
// ===== library: MasterCopy "Scale_current_output" =====

FUNCTION "Scale_current_output" : Void   // FC2, LAD
TITLE = Scale current output from 4-20 mA to 0-20 mA
{ S7_Optimized_Access := 'FALSE' }
VERSION : 0.1
// (27648-5530) 
// f(x) =  ------------------------- * x +5530 
//                 27648
   VAR_INPUT
      "r_output_4-20mA" : Real;
   END_VAR
   VAR_OUTPUT
      "w_output_0-20mA" : Word;
   END_VAR
   VAR_TEMP
      r_analog_ouput_temp : Real;
      r_factor : Real;
   END_VAR
BEGIN

REGION Network 1
   // multiply  by range  4-20mA ( 27648-5529,6=22118,4)
   // f(x1) = x * 22118
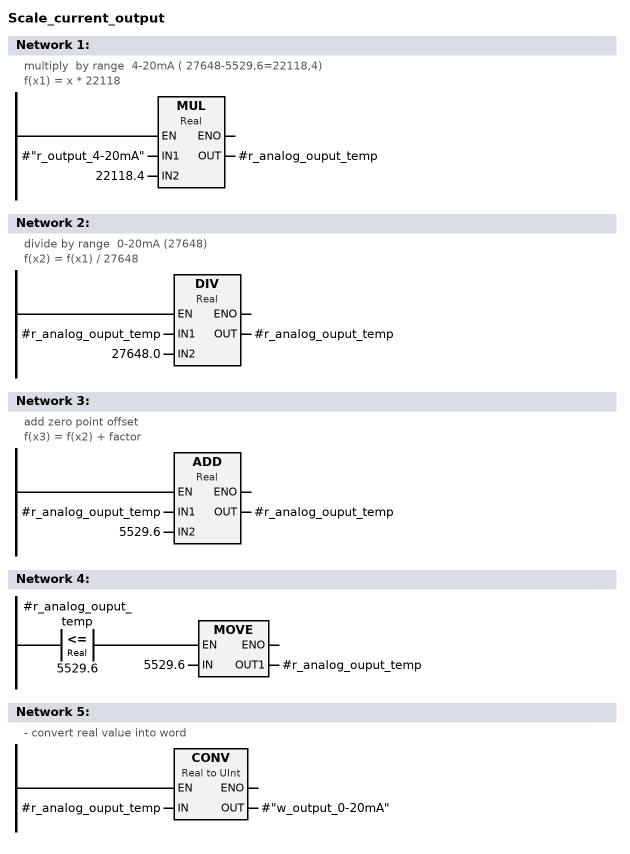
   RUNG wire#powerrail
      { S7_Templates := "SrcType := Real"; S7_GenerateENO := "TRUE" } Mul(in1 := #"r_output_4-20mA", in2 := 22118.4, out => #r_analog_ouput_temp)
   END_RUNG
   // the same network as SCL:
   #r_analog_ouput_temp := #"r_output_4-20mA" * 22118.4;
END_REGION

REGION Network 2
   // divide by range  0-20mA (27648)
   // f(x2) = f(x1) / 27648
   RUNG wire#powerrail
      { S7_Templates := "SrcType := Real"; S7_GenerateENO := "TRUE" } Div(in1 := #r_analog_ouput_temp, in2 := 27648.0, out => #r_analog_ouput_temp)
   END_RUNG
   // the same network as SCL:
   #r_analog_ouput_temp := #r_analog_ouput_temp / 27648.0;
END_REGION

REGION Network 3
   // add zero point offset
   // f(x3) = f(x2) + factor
   RUNG wire#powerrail
      { S7_Templates := "SrcType := Real"; S7_GenerateENO := "TRUE" } Add(in1 := #r_analog_ouput_temp, in2 := 5529.6, out => #r_analog_ouput_temp)
   END_RUNG
   // the same network as SCL:
   #r_analog_ouput_temp := #r_analog_ouput_temp + 5529.6;
END_REGION

REGION Network 4
   RUNG wire#powerrail
      { S7_Templates := "SrcType := Real" } LE_Contact(in1 := #r_analog_ouput_temp, in2 := 5529.6)
      { S7_GenerateENO := "TRUE" } Move(in := 5529.6, out1 => #r_analog_ouput_temp)
   END_RUNG
   // the same network as SCL:
   IF #r_analog_ouput_temp <= 5529.6 THEN #r_analog_ouput_temp := 5529.6; END_IF;
END_REGION

REGION Network 5
   // - convert real value into word
   RUNG wire#powerrail
      { S7_Templates := "[SrcType := Real, DestType := UInt]"; S7_GenerateENO := "TRUE" } Convert(in := #r_analog_ouput_temp, out => #"w_output_0-20mA")
   END_RUNG
   // the same network as SCL:
   #"w_output_0-20mA" := REAL_TO_UINT(#r_analog_ouput_temp);
END_REGION
END_FUNCTION

// ===== library: MasterCopy "Scale_current_input" =====

FUNCTION "Scale_current_input" : Void   // FC1, LAD
TITLE = Scale current input from 0-20 mA to 4-20 mA
{ S7_Optimized_Access := 'FALSE' }
VERSION : 0.1
// 27648
// f(x) =  ------------------------------- * x - 6912
//            (27648 - 5529,6)
   VAR_INPUT
      r_wire_break_limit : Real;
      "w_input_0-20mA" : Word;
   END_VAR
   VAR_OUTPUT
      b_wire_break : Bool;
      "r_input_4-20mA" : Real;
   END_VAR
   VAR_TEMP
      r_analog_input_temp : Real;
      r_factor : Real;
   END_VAR
   VAR_TEMP   // added for the SCL form of the ladder/FBD networks
      _w1 : Bool;
   END_VAR
BEGIN

REGION Network 1
   // - Convert analog  value to real
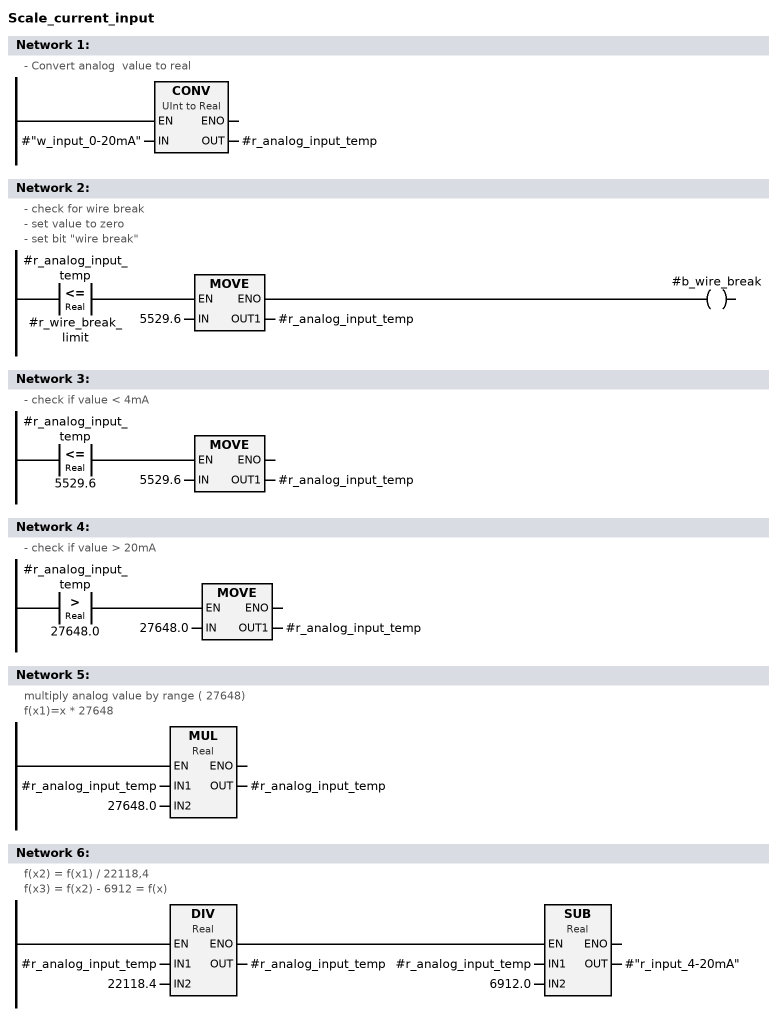
   RUNG wire#powerrail
      { S7_Templates := "[SrcType := UInt, DestType := Real]"; S7_GenerateENO := "TRUE" } Convert(in := #"w_input_0-20mA", out => #r_analog_input_temp)
   END_RUNG
   // the same network as SCL:
   #r_analog_input_temp := UINT_TO_REAL(#"w_input_0-20mA");
END_REGION

REGION Network 2
   // - check for wire break 
   //  - set value to zero
   //  - set bit "wire break"
   RUNG wire#powerrail
      { S7_Templates := "SrcType := Real" } LE_Contact(in1 := #r_analog_input_temp, in2 := #r_wire_break_limit)
      { S7_GenerateENO := "TRUE" } Move(in := 5529.6, out1 => #r_analog_input_temp)
      Coil( #b_wire_break )
   END_RUNG
   // the same network as SCL:
   // ENO of a box is taken as its EN; it also drops when the box reports an error
   #_w1 := #r_analog_input_temp <= #r_wire_break_limit;
   IF #_w1 THEN #r_analog_input_temp := 5529.6; END_IF;
   #b_wire_break := #_w1;
END_REGION

REGION Network 3
   // - check if value < 4mA
   RUNG wire#powerrail
      { S7_Templates := "SrcType := Real" } LE_Contact(in1 := #r_analog_input_temp, in2 := 5529.6)
      { S7_GenerateENO := "TRUE" } Move(in := 5529.6, out1 => #r_analog_input_temp)
   END_RUNG
   // the same network as SCL:
   IF #r_analog_input_temp <= 5529.6 THEN #r_analog_input_temp := 5529.6; END_IF;
END_REGION

REGION Network 4
   // - check if value > 20mA
   RUNG wire#powerrail
      { S7_Templates := "SrcType := Real" } GT_Contact(in1 := #r_analog_input_temp, in2 := 27648.0)
      { S7_GenerateENO := "TRUE" } Move(in := 27648.0, out1 => #r_analog_input_temp)
   END_RUNG
   // the same network as SCL:
   IF #r_analog_input_temp > 27648.0 THEN #r_analog_input_temp := 27648.0; END_IF;
END_REGION

REGION Network 5
   // multiply analog value by range ( 27648)
   // f(x1)=x * 27648
   RUNG wire#powerrail
      { S7_Templates := "SrcType := Real"; S7_GenerateENO := "TRUE" } Mul(in1 := #r_analog_input_temp, in2 := 27648.0, out => #r_analog_input_temp)
   END_RUNG
   // the same network as SCL:
   #r_analog_input_temp := #r_analog_input_temp * 27648.0;
END_REGION

REGION Network 6
   // f(x2) = f(x1) / 22118,4
   // f(x3) = f(x2) - 6912 = f(x)
   RUNG wire#powerrail
      { S7_Templates := "SrcType := Real"; S7_GenerateENO := "TRUE" } Div(in1 := #r_analog_input_temp, in2 := 22118.4, out => #r_analog_input_temp)
      { S7_Templates := "SrcType := Real"; S7_GenerateENO := "TRUE" } Sub(in1 := #r_analog_input_temp, in2 := 6912.0, out => #"r_input_4-20mA")
   END_RUNG
   // the same network as SCL:
   // ENO of a box is taken as its EN; it also drops when the box reports an error
   #r_analog_input_temp := #r_analog_input_temp / 22118.4;
   #"r_input_4-20mA" := #r_analog_input_temp - 6912.0;
END_REGION
END_FUNCTION